(* PLC project Unnamed, Unknown Unnamed 1 *)
(* stored: creationDateTime 2024-05-09T12:14:32, modificationDateTime 2024-11-01T19:16:07 *)

PROGRAM READ_WRITE_EXAMPLE
  VAR
    BLINK AT %QX0.0 : BOOL := false;  (* description 0 *)
  END_VAR
  VAR
    CONF_FLAG : BOOL := false;  (* description 1 *)
    WRITE_DONE_FLAG : BOOL := false;  (* description 2 *)
    READ_DONE_FLAG : BOOL := false;  (* description 3 *)
    BIT_RATE : LINT := 250000;  (* description 4 *)
    CHANNEL : USINT := 1;  (* description 5 *)
    ID : DWORD := 16#18FF3900;
    ID_READ : DWORD;
    D0 : BYTE := 16#01;
    D1 : BYTE := 16#02;
    D2 : BYTE := 16#03;
    D3 : BYTE := 16#12;
    D4 : BYTE := 16#3D;
    D5 : BYTE := 16#4A;
    D6 : BYTE := 16#A2;
    D7 : BYTE := 16#C3;
    D0_READ : BYTE;
    D1_READ : BYTE;
    D2_READ : BYTE;
    D3_READ : BYTE;
    D4_READ : BYTE;
    D5_READ : BYTE;
    D6_READ : BYTE;
    D7_READ : BYTE;
    TOF0 : TOF;
    TON0 : TON;
    STM32CAN_CONF0 : STM32CAN_CONF;
    R_TRIG1 : R_TRIG;
    STM32CAN_WRITE0 : STM32CAN_WRITE;
    STM32CAN_READ0 : STM32CAN_READ;
    R_TRIG7 : R_TRIG;
    STM32CAN_WRITE6 : STM32CAN_WRITE;
  END_VAR

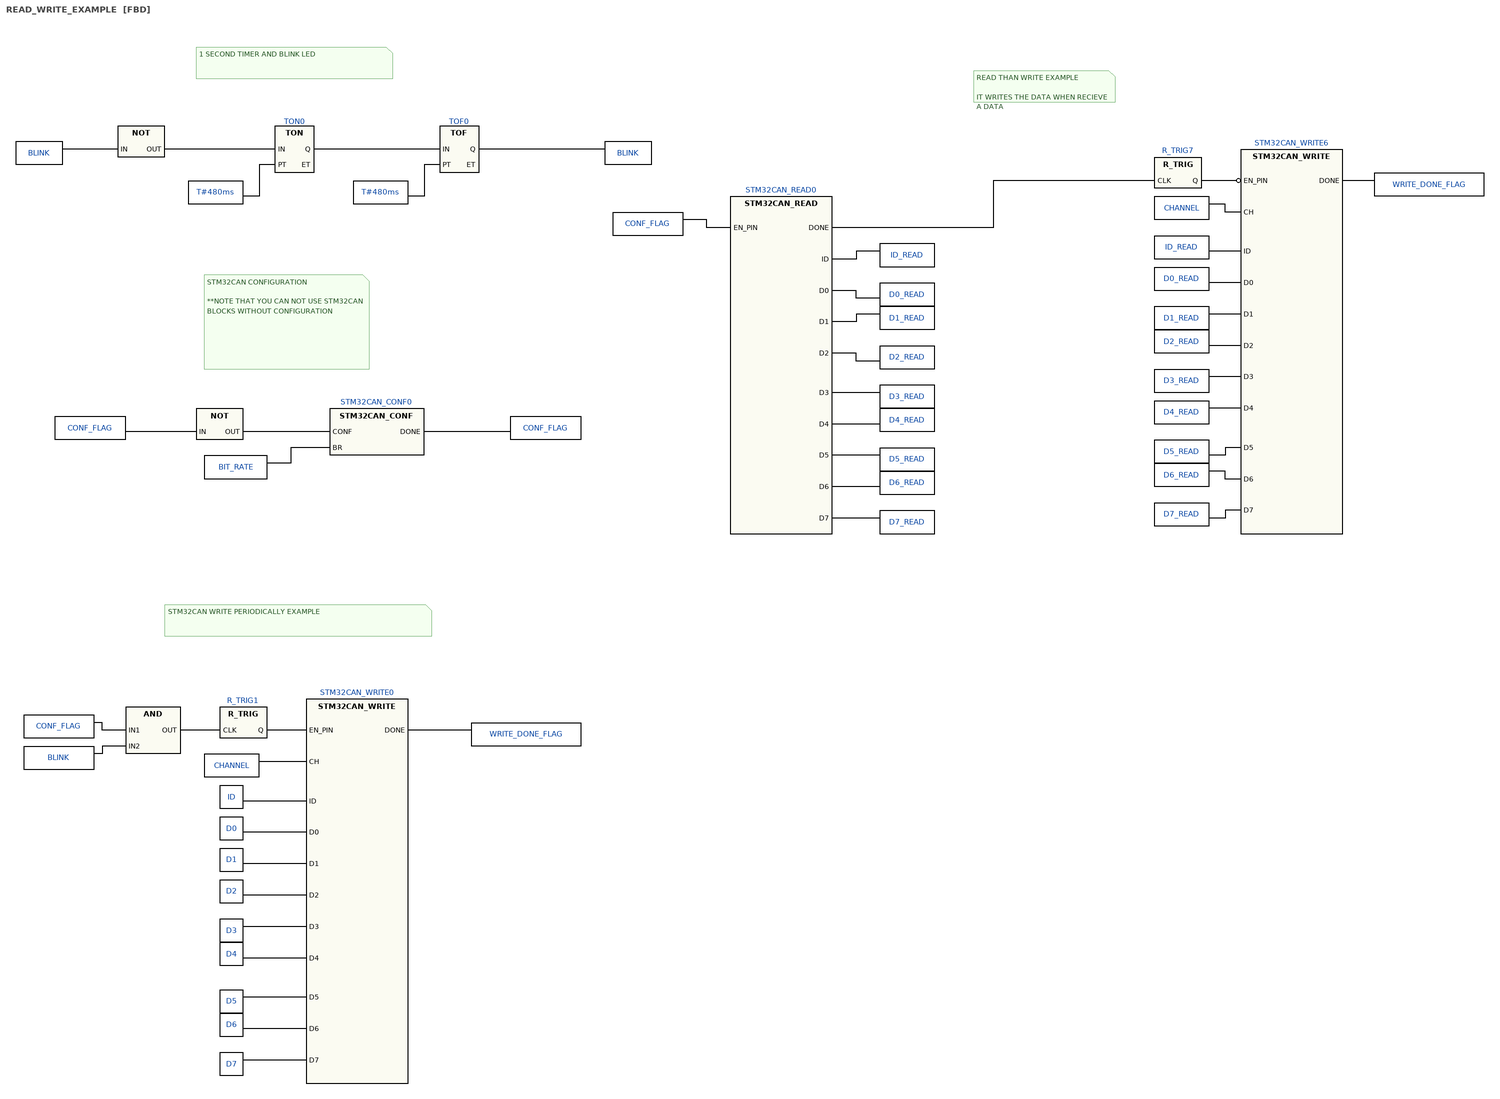
(* FBD diagram, written out as Structured Text *)
(* 1 SECOND TIMER AND BLINK LED *)
(* READ THAN WRITE EXAMPLE

IT WRITES THE DATA WHEN RECIEVE A DATA *)
TON0(IN := NOT BLINK, PT := T#480ms);
TOF0(IN := TON0.Q, PT := T#480ms);
BLINK := TOF0.Q;
(* STM32CAN CONFIGURATION

**NOTE THAT YOU CAN NOT USE STM32CAN BLOCKS WITHOUT CONFIGURATION *)
(* STM32CAN WRITE PERIODICALLY EXAMPLE *)
R_TRIG1(CLK := CONF_FLAG AND BLINK);
STM32CAN_WRITE0(EN_PIN := R_TRIG1.Q, CH := CHANNEL, ID := ID, D0 := D0, D1 := D1, D2 := D2, D3 := D3, D4 := D4, D5 := D5, D6 := D6, D7 := D7);
WRITE_DONE_FLAG := STM32CAN_WRITE0.DONE;
STM32CAN_CONF0(CONF := NOT CONF_FLAG, BR := BIT_RATE);
CONF_FLAG := STM32CAN_CONF0.DONE;
STM32CAN_READ0(EN_PIN := CONF_FLAG);
ID_READ := STM32CAN_READ0.ID;
D0_READ := STM32CAN_READ0.D0;
D1_READ := STM32CAN_READ0.D1;
D2_READ := STM32CAN_READ0.D2;
D3_READ := STM32CAN_READ0.D3;
D4_READ := STM32CAN_READ0.D4;
D5_READ := STM32CAN_READ0.D5;
D6_READ := STM32CAN_READ0.D6;
D7_READ := STM32CAN_READ0.D7;
R_TRIG7(CLK := STM32CAN_READ0.DONE);
STM32CAN_WRITE6(EN_PIN := NOT R_TRIG7.Q, CH := CHANNEL, ID := ID_READ, D0 := D0_READ, D1 := D1_READ, D2 := D2_READ, D3 := D3_READ, D4 := D4_READ, D5 := D5_READ, D6 := D6_READ, D7 := D7_READ);
WRITE_DONE_FLAG := STM32CAN_WRITE6.DONE;
END_PROGRAM

CONFIGURATION Config0
  RESOURCE Res0 ON PLC
    TASK task0(INTERVAL := T#20ms, PRIORITY := 0);
    PROGRAM instance0 WITH task0 : READ_WRITE_EXAMPLE;
  END_RESOURCE
END_CONFIGURATION
